(* CODESYS project controllerClass3.project

Project tree, tasks and I/O mapping:
  Device : Elmo Platinum Maestro, Elmo Motion Control, version 1.0.0.2
    application Application
      libraries: Standard, * (System); VisuDialogs, * (System)
      task MainTask (cyclic, interval t#20ms, priority 1) calls PLC_PRG
      task VISU_TASK (cyclic, interval 100 ms, priority 31) calls VisuElems.Visu_Prg
      program PLC_PRG [ST]
      01_Enumerator/
      02_Structure/
        data type stCar
      03_Module/
        function block FB_Car [ST]: M_CalcDist, M_CalcRefuel, pFuel, pModel, M_LightCtrl
        function block FB_CarAdv [ST]: M_LightCtrl, pModel
      visualisation Car
      visualisation Visualization
      04_Component/
        interface ITF_LightCtrl: M_ON, M_OFF
        function block FB_LightONOFF [ST]: M_ON, M_OFF
        function block FB_LightDimm [ST]: M_ON, M_OFF
    Elmo_Master_Device : Elmo Master Device, Elmo, version 1.0.0.2
  libraries: VisuSymbols, 3.5.10.0 (System)
  text list GlobalTextList
*)

// Device/Application/02_Structure/stCar
TYPE stCar :
STRUCT
	xKey : BOOL;
	iMeters: INT;
	sStatus: STRING;
	
	uiSetFuel : UINT;
	uiGetFuel : UINT;
	
	xRefuel: BOOL;
	trig_Refuel: r_trig;
	
	sModel: STRING;
	
	xTypeNormal: BOOL:= TRUE;
	xLightON: BOOL;
	uiLightIntensity: UINT;
	
END_STRUCT
END_TYPE

// Device/Application/PLC_PRG
PROGRAM PLC_PRG
VAR
	fbCar: ARRAY [1..uiObject] OF FB_Car;
	//xKey: BOOL;
	//iMeters: INT;
	//uiFuel: UINT;
	stCarData : ARRAY [1..uiObject] OF stCar;
	iCnt: INT;
	fbCarAdv: FB_CarAdv;
	stCarAdvData : stCar;
END_VAR

VAR CONSTANT
	uiObject: UINT:= 3;
END_VAR

//fbCar.ix_Start := xKey;

//iMeters := fbCar.M_CalcDist();

//uiFuel := fbCar.M_CalcRefuel();

FOR iCnt:= 1 TO uiObject BY 1 DO
    stCarData[iCnt].sModel := fbCar[iCnt].pModel;	

	fbCar[iCnt].ix_Start := stCarData[iCnt].xKey;
	stCarData[iCnt].iMeters := fbCar[iCnt].M_CalcDist();
	stCarData[iCnt].sStatus := fbCar[iCnt].os_Status;
	
	stCarData[iCnt].trig_Refuel (clk := stCarData[iCnt].xRefuel);
	IF stCarData[iCnt].trig_Refuel.Q THEN
		fbCar[iCnt].pFuel := stCarData[iCnt].uiSetFuel;
	END_IF
	stCarData[iCnt].uiGetFuel := fbCar[iCnt].pFuel;
	
	stCarData[iCnt].uiLightIntensity := fbCar[iCnt].M_LightCtrl(stCarData[iCnt].xTypeNormal,stCarData[iCnt].xLightON);
END_FOR


stCarAdvData.sModel := fbCarAdv.pModel;	

	fbCarAdv.ix_Start := stCarAdvData.xKey;
	stCarAdvData.iMeters := fbCarAdv.M_CalcDist();
	stCarAdvData.sStatus := fbCarAdv.os_Status;
	
	stCarAdvData.trig_Refuel (clk := stCarAdvData.xRefuel);
	IF stCarAdvData.trig_Refuel.Q THEN
		fbCarAdv.pFuel := stCarAdvData.uiSetFuel;
	END_IF
	stCarAdvData.uiGetFuel := fbCarAdv.pFuel;
	
	stCarAdvData.uiLightIntensity := fbCarAdv.M_LightCtrl(stCarAdvData.xTypeNormal,stCarAdvData.xLightON);

END_PROGRAM

// Device/Application/03_Module/FB_Car
FUNCTION_BLOCK FB_Car
VAR_INPUT
	ix_Start: BOOL;
END_VAR
VAR_OUTPUT
	os_Status: STRING;
END_VAR
VAR
	iMove: INT;
	uiFuel: UINT := 1000;
	sModel: STRING;
	
	fbLightONOFF : FB_LightONOFF;
	fbLightDimm : FB_LightDimm;
	itfLightCtrl: ITF_LightCtrl;
END_VAR

METHOD M_CalcDist : INT
VAR_INPUT
END_VAR
IF ix_Start THEN
	iMove := iMove + 1;
	M_CalcDist := iMove/100;
	M_CalcRefuel();
	os_Status := 'Moving';
ELSE
	os_Status := 'Stopped';
END_IF
END_METHOD

METHOD PRIVATE M_CalcRefuel : UINT
VAR_INPUT
END_VAR
IF (iMove MOD 100) = 0 THEN
	uiFuel := uiFuel - 10;
END_IF
END_METHOD

PROPERTY pFuel : UINT
SET
IF (pFuel + uiFuel) > 4000 THEN
	uiFuel := 4000;
ELSIF pFuel < 0 THEN
	uiFuel := 0;
ELSE
	uiFuel := pFuel + uiFuel;
END_IF
END_SET
GET
IF uiFuel <= 0 THEN
	pFuel := 0;
ELSE
	pFuel := uiFuel;
END_IF
END_GET
END_PROPERTY

PROPERTY pModel : STRING
GET
pModel := 'Focus';
END_GET
END_PROPERTY

METHOD M_LightCtrl : UINT
VAR_INPUT
	xTypeNormal: BOOL;
	xLightON: bool;
END_VAR
IF xTypeNormal THEN
	itfLightCtrl := fbLightONOFF;
ELSE
	itfLightCtrl := fbLightDimm;
END_IF

IF xLightON THEN
	M_LightCtrl := itfLightCtrl.M_ON();
ELSE
	M_LightCtrl := itfLightCtrl.M_OFF();
END_IF
END_METHOD

END_FUNCTION_BLOCK

// Device/Application/04_Component/FB_LightONOFF
FUNCTION_BLOCK FB_LightONOFF IMPLEMENTS ITF_LightCtrl
VAR_INPUT
END_VAR
VAR_OUTPUT
END_VAR
VAR
	uiLight: UINT;
END_VAR

{warning 'add method implementation'}
METHOD M_ON : UINT
uiLight := 100;
M_ON := uiLight;
END_METHOD

{warning 'add method implementation'}
METHOD M_OFF : UINT
uiLight := 0;
M_OFF := uiLight;
END_METHOD

END_FUNCTION_BLOCK

// Device/Application/04_Component/ITF_LightCtrl
INTERFACE ITF_LightCtrl

METHOD M_ON : UINT
VAR_INPUT
END_VAR
END_METHOD

METHOD M_OFF : UINT
VAR_INPUT
END_VAR
END_METHOD

END_INTERFACE

// Device/Application/04_Component/FB_LightDimm
FUNCTION_BLOCK FB_LightDimm IMPLEMENTS ITF_LightCtrl
VAR_INPUT
END_VAR
VAR_OUTPUT
END_VAR
VAR
	uiLight: UINT;
	uiInc: UINT:=5;
END_VAR

{warning 'add method implementation'}
METHOD M_ON : UINT
IF uiLight < 100 THEN
	uiLight := uiLight + uiInc;
ELSE
	uiLight := 100;
END_IF

M_ON := uiLight;
END_METHOD

{warning 'add method implementation'}
METHOD M_OFF : UINT
IF uiLight > 0 THEN
	uiLight := uiLight - uiInc;
ELSE
	uiLight := 0;
END_IF

M_OFF := uiLight;
END_METHOD

END_FUNCTION_BLOCK

// Device/Application/03_Module/FB_CarAdv
FUNCTION_BLOCK FB_CarAdv EXTENDS FB_Car
VAR_INPUT
END_VAR
VAR_OUTPUT
END_VAR
VAR
END_VAR

SUPER^();

METHOD M_LightCtrl : UINT
VAR_INPUT
	xTypeNormal: BOOL;
	xLightON: bool;
END_VAR
itfLightCtrl:= fbLightDimm;

IF xLightON THEN
	M_LightCtrl := itfLightCtrl.M_ON();
ELSE
	M_LightCtrl := itfLightCtrl.M_OFF();
END_IF
END_METHOD

PROPERTY pModel : STRING
GET
pModel := CONCAT(STR1 := SUPER^.pModel, STR2 := 'ADV');
END_GET
END_PROPERTY

END_FUNCTION_BLOCK

// Device/Application/Car
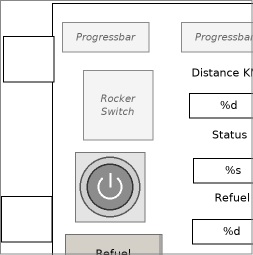
VISUALIZATION Car  // 253x255
VAR_IN_OUT
	stCarVisu: stCar;
END_VAR
    RoundedRectangle (52,3 234x329)
    Rectangle (285,204 51x46)
    Rectangle (284,37 51x46)
    Rectangle (3,36 51x46)
    Rectangle (1,196 51x46)
    Rectangle (193,158 80x25), "%s", text variable: stCarVisu.sStatus
    Rectangle (189,93 80x25), "%d", text variable: stCarVisu.iMeters
    PowerSwitch (75,152 70x70), variable: stCarVisu.xKey, behaviour: TOGGLE, style: Switch-PowerSwitch-Gray
    Label (181,58 89x30), "Distance KM"
    Label (185,120 89x30), "Status"
    Label (188,183 89x30), "Refuel"
    Rectangle (192,219 80x25), "%d", text variable: stCarVisu.uiSetFuel
        OnMouseClick: write the text variable via VisuDialogs.Numpad
    Rectangle (188,285 80x25), "%d", text variable: stCarVisu.uiGetFuel
    Label (186,245 89x30), "Current Fuel"
    Button (65,234 97x40), "Refuel"
        tap stCarVisu.xRefuel
    RockerSwitch (83,70 70x70), variable: stCarVisu.xLightON, behaviour: TOGGLE, style: Switch-RockerSwitch-Gray
    Progressbar (62,22 87x30), variable: stCarVisu.uiLightIntensity
    Progressbar (181,22 87x30), variable: stCarVisu.uiLightIntensity
    Rectangle (128,333 150x30), "%s", text variable: stCarVisu.sModel
    Label (32,333 88x30), "Model"
END_VISUALIZATION

// Device/Application/Visualization
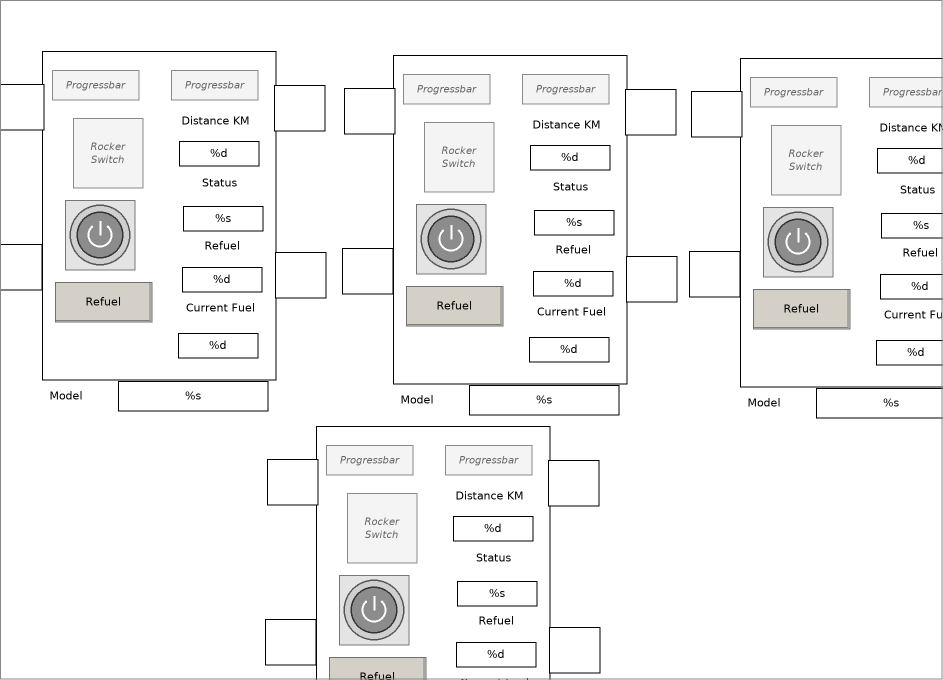
VISUALIZATION Visualization  // 943x680
    Frame (-10,48 253x255)
        shows Car(stCarVisu := PLC_PRG.stCarData[1])
    Frame (341,52 253x255)
        shows Car(stCarVisu := PLC_PRG.stCarData[2])
    Frame (688,55 253x255)
        shows Car(stCarVisu := PLC_PRG.stCarData[3])
    Frame (264,423 253x255)
        shows Car(stCarVisu := PLC_PRG.stCarAdvData)
END_VISUALIZATION
